{attribute 'GeneratedUsingTerminal: EL3443-0000-0016'}
{attribute addProperty BoxType "EL3443-0000-0016"}
{attribute addProperty Id "Voltage_Sign_BitAT %I*BOOL1OvervoltageAT %I*BOOL1OvercurrentAT %I*BOOL1Inaccurate_VoltageAT %I*BOOL1Inaccurate_CurrentAT %I*BOOL1Voltage_Guard_WarningAT %I*BOOL1Voltage_Guard_ErrorAT %I*BOOL1Current_Guard_WarningAT %I*BOOL1Current_Guard_ErrorAT %I*BOOL1TxPDO_ToggleAT %I*BOOL1"}
{attribute addProperty CRC "1639876758"}
{attribute addProperty Size "10"}
TYPE L1_Status_61BE8896 :
STRUCT
	{attribute addProperty Name "Voltage_Sign_Bit"}
	Voltage_Sign_Bit AT %I* : BOOL;
	{attribute addProperty Name "Overvoltage"}
	Overvoltage AT %I* : BOOL;
	{attribute addProperty Name "Overcurrent"}
	Overcurrent AT %I* : BOOL;
	{attribute addProperty Name "Inaccurate_Voltage"}
	Inaccurate_Voltage AT %I* : BOOL;
	{attribute addProperty Name "Inaccurate_Current"}
	Inaccurate_Current AT %I* : BOOL;
	{attribute addProperty Name "Voltage_Guard_Warning"}
	Voltage_Guard_Warning AT %I* : BOOL;
	{attribute addProperty Name "Voltage_Guard_Error"}
	Voltage_Guard_Error AT %I* : BOOL;
	{attribute addProperty Name "Current_Guard_Warning"}
	Current_Guard_Warning AT %I* : BOOL;
	{attribute addProperty Name "Current_Guard_Error"}
	Current_Guard_Error AT %I* : BOOL;
	{attribute addProperty Name "TxPDO_Toggle"}
	TxPDO_Toggle AT %I* : BOOL;
END_STRUCT
END_TYPE

(* stored: Version 1.2.0.0, ProductVersion 3.1.4024.9
   DUT L1_Status_61BE8896: Id {d8bad7d1-735a-496d-be8f-f8461a311367} *)
